FUNCTION "WL_2WordToDint" : DInt
{ S7_Optimized_Access := 'TRUE' }
VERSION : 0.1
   VAR_INPUT
      Word0 : Word;
      Word1 : Word;
   END_VAR

   VAR_TEMP
      tempDword : DWord;
   END_VAR


BEGIN
	#tempDword.%W0 := #Word0;
	#tempDword.%W1 := #Word1;

	#WL_2WordToDint := DWORD_TO_DINT(#tempDword);
END_FUNCTION

